// TIA Portal V19 export
DATA_BLOCK "MB_MASTER_DB"   // DB55
// stored: InstanceOfName MB_MASTER, OfSystemLibElement MB_MASTER, OfSystemLibVersion 2.2
"MB_MASTER"
   // // inherited from MB_BASE
   // VAR_INPUT
   //    REQ : Bool;
   //    MB_ADDR : UInt;
   //    MODE : USInt;
   //    DATA_ADDR : UDInt;
   //    DATA_LEN : UInt;
   // END_VAR
   // VAR_OUTPUT
   //    DONE : Bool;
   //    BUSY : Bool;
   //    ERROR : Bool;
   //    STATUS : Word;
   // END_VAR
   // VAR_IN_OUT
   //    DATA_PTR : Variant;
   // END_VAR
   // VAR
   //    SEND_PTP_SFB : Array[0..11] of Byte;
   //    RCV_PTP_SFB : Array[0..11] of Byte;
   //    RCV_RST_SFB : Array[0..9] of Byte;
   //    PF_FREQUENCY : Real;
   //    BLOCKED_PROC_TIMEOUT : Real;
   //    CURRENT_TIME_VALUE : UDInt;
   //    SAVED_TIME_VALUE : UDInt;
   //    SAVED_SLAVE_ADDR : Word;
   //    SAVED_MODE : Word;
   //    SAVED_DATA_ADDR : DWord;
   //    SAVED_DATA_LEN : UInt;
   //    MB_STATE : UInt;
   //    COMM_SENT_COUNT : UInt;
   //    BYTE_COUNT : USInt;
   //    INIT_OK : Bool;
   //    ACTIVE : Bool;
   //    BROADCAST_FLAG : Bool;
   //    EXTENDED_ADDRESSING : Bool;
   //    SAVED_START_ADDR : UInt;
   //    TXBuf_Function_Offset : UDInt;
   //    TXBuf_Address_Offset : UDInt;
   //    TXBuf_Quantity_Offset : UDInt;
   // END_VAR
BEGIN
END_DATA_BLOCK
